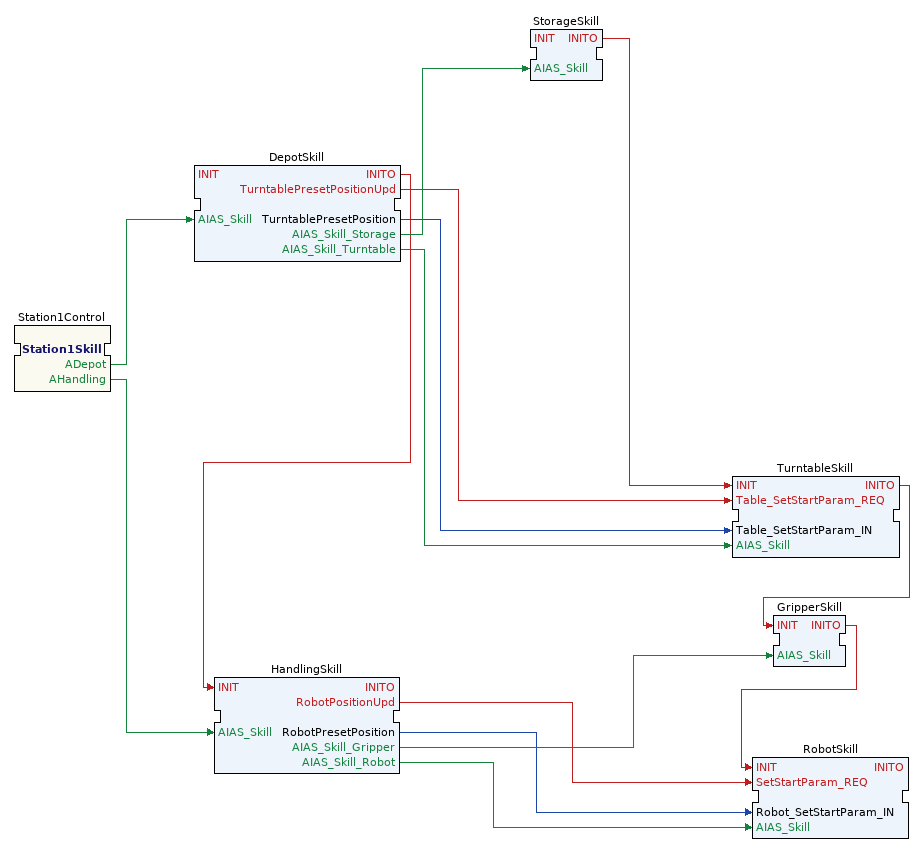
    [picture p24: application VDMA_Station1_SkillbasedControl]
    FBS
      Station1Control : Station1Skill;
    END_FBS
    SUBAPPLICATION StorageSkill
      EVENT_INPUT
        INIT;
      END_EVENT
      EVENT_OUTPUT
        INITO;
      END_EVENT
      SOCKETS
        AIAS_Skill : IAS_Skill;
      END_SOCKETS
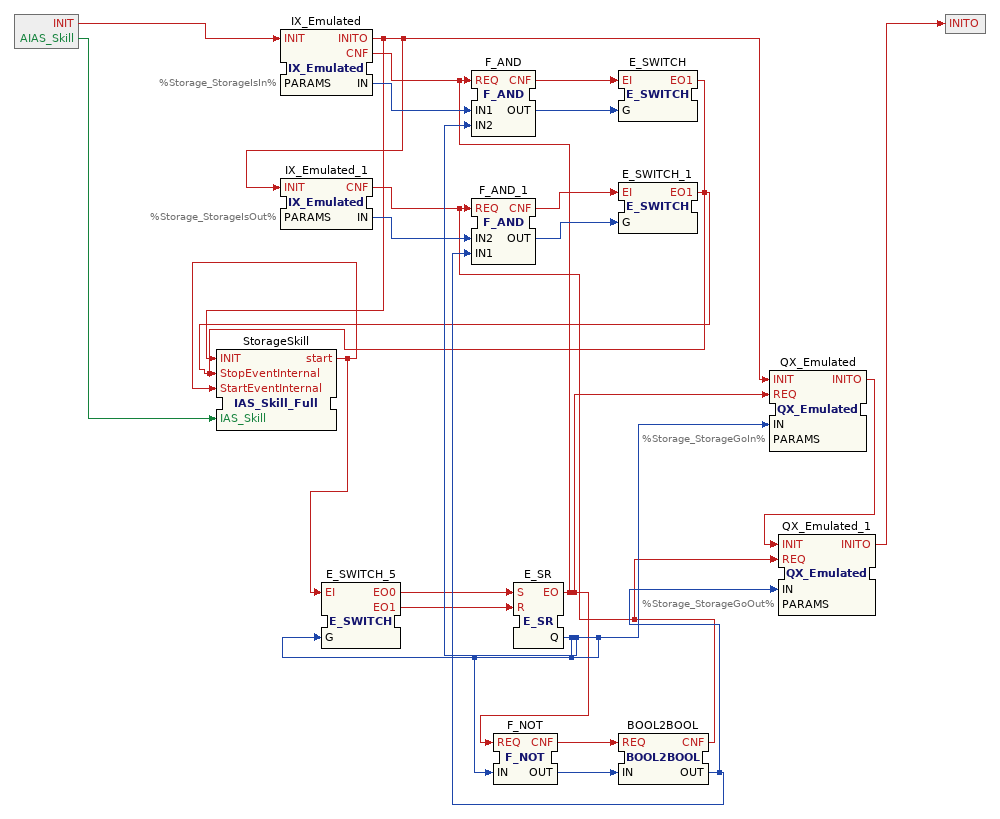
      FBS
        E_SWITCH_5 : E_SWITCH;
        IX_Emulated : IX_Emulated(PARAMS := %Storage_StorageIsIn%);
        F_NOT : F_NOT;
        IX_Emulated_1 : IX_Emulated(PARAMS := %Storage_StorageIsOut%);
        E_SWITCH : E_SWITCH;
        E_SWITCH_1 : E_SWITCH;
        StorageSkill : IAS_Skill_Full;
        F_AND : F_AND;
        BOOL2BOOL : BOOL2BOOL;
        F_AND_1 : F_AND;
        E_SR : E_SR;
        QX_Emulated_1 : QX_Emulated(PARAMS := %Storage_StorageGoOut%);
        QX_Emulated : QX_Emulated(PARAMS := %Storage_StorageGoIn%);
      END_FBS
      EVENT_CONNECTIONS
        StorageSkill.start TO E_SWITCH_5.EI;
        E_SWITCH_5.EO0 TO E_SR.S;
        E_SWITCH_5.EO1 TO E_SR.R;
        IX_Emulated.INITO TO IX_Emulated_1.INIT;
        IX_Emulated.INITO TO StorageSkill.INIT;
        IX_Emulated.CNF TO F_AND.REQ;
        E_SR.EO TO F_NOT.REQ;
        F_NOT.CNF TO BOOL2BOOL.REQ;
        IX_Emulated_1.CNF TO F_AND_1.REQ;
        F_AND.CNF TO E_SWITCH.EI;
        E_SWITCH.EO1 TO StorageSkill.StopEventInternal;
        F_AND_1.CNF TO E_SWITCH_1.EI;
        E_SWITCH_1.EO1 TO StorageSkill.StopEventInternal;
        StorageSkill.start TO StorageSkill.StartEventInternal;
        E_SR.EO TO F_AND.REQ;
        BOOL2BOOL.CNF TO F_AND_1.REQ;
        INIT TO IX_Emulated.INIT;
        QX_Emulated_1.INITO TO INITO;
        IX_Emulated.INITO TO QX_Emulated.INIT;
        QX_Emulated.INITO TO QX_Emulated_1.INIT;
        BOOL2BOOL.CNF TO QX_Emulated_1.REQ;
        E_SR.EO TO QX_Emulated.REQ;
      END_CONNECTIONS
      DATA_CONNECTIONS
        E_SR.Q TO E_SWITCH_5.G;
        IX_Emulated.IN TO F_AND.IN1;
        E_SR.Q TO F_NOT.IN;
        F_NOT.OUT TO BOOL2BOOL.IN;
        IX_Emulated_1.IN TO F_AND_1.IN2;
        F_AND.OUT TO E_SWITCH.G;
        F_AND_1.OUT TO E_SWITCH_1.G;
        E_SR.Q TO F_AND.IN2;
        BOOL2BOOL.OUT TO F_AND_1.IN1;
        E_SR.Q TO QX_Emulated.IN;
        BOOL2BOOL.OUT TO QX_Emulated_1.IN;
      END_CONNECTIONS
      ADAPTER_CONNECTIONS
        AIAS_Skill TO StorageSkill.IAS_Skill;
      END_CONNECTIONS
    END_SUBAPPLICATION
    SUBAPPLICATION TurntableSkill
      EVENT_INPUT
        INIT;
        Table_SetStartParam_REQ;
      END_EVENT
      EVENT_OUTPUT
        INITO;
      END_EVENT
      VAR_INPUT
        Table_SetStartParam_IN : WORD;
      END_VAR
      SOCKETS
        AIAS_Skill : IAS_Skill;
      END_SOCKETS
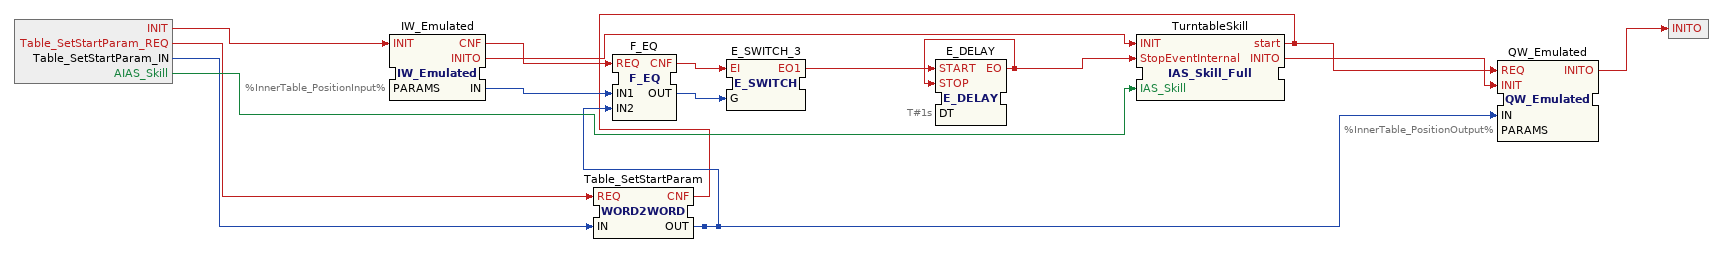
      FBS
        F_EQ : F_EQ;
        E_SWITCH_3 : E_SWITCH;
        Table_SetStartParam : WORD2WORD;
        QW_Emulated : QW_Emulated(PARAMS := %InnerTable_PositionOutput%);
        TurntableSkill : IAS_Skill_Full;
        IW_Emulated : IW_Emulated(PARAMS := %InnerTable_PositionInput%);
        E_DELAY : E_DELAY(DT := T#1s);
      END_FBS
      EVENT_CONNECTIONS
        IW_Emulated.CNF TO F_EQ.REQ;
        TurntableSkill.start TO F_EQ.REQ;
        Table_SetStartParam.CNF TO F_EQ.REQ;
        F_EQ.CNF TO E_SWITCH_3.EI;
        TurntableSkill.start TO QW_Emulated.REQ;
        Table_SetStartParam_REQ TO Table_SetStartParam.REQ;
        INIT TO IW_Emulated.INIT;
        IW_Emulated.INITO TO TurntableSkill.INIT;
        TurntableSkill.INITO TO QW_Emulated.INIT;
        QW_Emulated.INITO TO INITO;
        E_SWITCH_3.EO1 TO E_DELAY.START;
        E_DELAY.EO TO TurntableSkill.StopEventInternal;
        E_DELAY.EO TO E_DELAY.STOP;
      END_CONNECTIONS
      DATA_CONNECTIONS
        IW_Emulated.IN TO F_EQ.IN1;
        Table_SetStartParam.OUT TO F_EQ.IN2;
        F_EQ.OUT TO E_SWITCH_3.G;
        Table_SetStartParam.OUT TO QW_Emulated.IN;
        Table_SetStartParam_IN TO Table_SetStartParam.IN;
      END_CONNECTIONS
      ADAPTER_CONNECTIONS
        AIAS_Skill TO TurntableSkill.IAS_Skill;
      END_CONNECTIONS
    END_SUBAPPLICATION
    SUBAPPLICATION DepotSkill
      EVENT_INPUT
        INIT;
      END_EVENT
      EVENT_OUTPUT
        INITO;
        TurntablePresetPositionUpd;
      END_EVENT
      VAR_OUTPUT
        TurntablePresetPosition : WORD;
      END_VAR
      SOCKETS
        AIAS_Skill : IAS_Skill;
      END_SOCKETS
      PLUGS
        AIAS_Skill_Storage : IAS_Skill;
        AIAS_Skill_Turntable : IAS_Skill;
      END_PLUGS
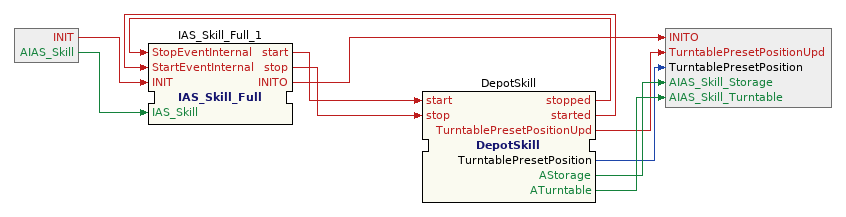
      FBS
        IAS_Skill_Full_1 : IAS_Skill_Full;
        DepotSkill : DepotSkill;
      END_FBS
      EVENT_CONNECTIONS
        DepotSkill.stopped TO IAS_Skill_Full_1.StopEventInternal;
        DepotSkill.started TO IAS_Skill_Full_1.StartEventInternal;
        IAS_Skill_Full_1.start TO DepotSkill.start;
        IAS_Skill_Full_1.stop TO DepotSkill.stop;
        DepotSkill.TurntablePresetPositionUpd TO TurntablePresetPositionUpd;
        INIT TO IAS_Skill_Full_1.INIT;
        IAS_Skill_Full_1.INITO TO INITO;
      END_CONNECTIONS
      DATA_CONNECTIONS
        DepotSkill.TurntablePresetPosition TO TurntablePresetPosition;
      END_CONNECTIONS
      ADAPTER_CONNECTIONS
        AIAS_Skill TO IAS_Skill_Full_1.IAS_Skill;
        DepotSkill.AStorage TO AIAS_Skill_Storage;
        DepotSkill.ATurntable TO AIAS_Skill_Turntable;
      END_CONNECTIONS
    END_SUBAPPLICATION
    SUBAPPLICATION GripperSkill
      EVENT_INPUT
        INIT;
      END_EVENT
      EVENT_OUTPUT
        INITO;
      END_EVENT
      SOCKETS
        AIAS_Skill : IAS_Skill;
      END_SOCKETS
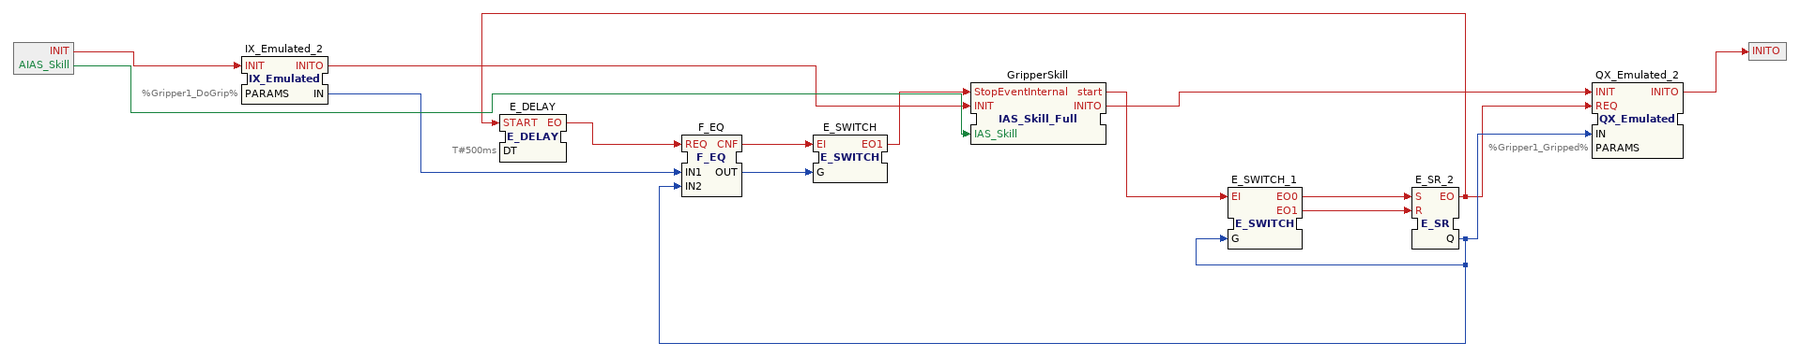
      FBS
        GripperSkill : IAS_Skill_Full;
        F_EQ : F_EQ;
        E_SWITCH_1 : E_SWITCH;
        IX_Emulated_2 : IX_Emulated(PARAMS := %Gripper1_DoGrip%);
        E_DELAY : E_DELAY(DT := T#500ms);
        E_SWITCH : E_SWITCH;
        E_SR_2 : E_SR;
        QX_Emulated_2 : QX_Emulated(PARAMS := %Gripper1_Gripped%);
      END_FBS
      EVENT_CONNECTIONS
        E_SWITCH.EO1 TO GripperSkill.StopEventInternal;
        GripperSkill.start TO E_SWITCH_1.EI;
        E_DELAY.EO TO F_EQ.REQ;
        F_EQ.CNF TO E_SWITCH.EI;
        E_SWITCH_1.EO0 TO E_SR_2.S;
        E_SWITCH_1.EO1 TO E_SR_2.R;
        E_SR_2.EO TO E_DELAY.START;
        INIT TO IX_Emulated_2.INIT;
        IX_Emulated_2.INITO TO GripperSkill.INIT;
        GripperSkill.INITO TO QX_Emulated_2.INIT;
        QX_Emulated_2.INITO TO INITO;
        E_SR_2.EO TO QX_Emulated_2.REQ;
      END_CONNECTIONS
      DATA_CONNECTIONS
        IX_Emulated_2.IN TO F_EQ.IN1;
        E_SR_2.Q TO F_EQ.IN2;
        F_EQ.OUT TO E_SWITCH.G;
        E_SR_2.Q TO E_SWITCH_1.G;
        E_SR_2.Q TO QX_Emulated_2.IN;
      END_CONNECTIONS
      ADAPTER_CONNECTIONS
        AIAS_Skill TO GripperSkill.IAS_Skill;
      END_CONNECTIONS
    END_SUBAPPLICATION
    SUBAPPLICATION HandlingSkill
      EVENT_INPUT
        INIT;
      END_EVENT
      EVENT_OUTPUT
        INITO;
        RobotPositionUpd;
      END_EVENT
      VAR_OUTPUT
        RobotPresetPosition : WORD;
      END_VAR
      SOCKETS
        AIAS_Skill : IAS_Skill;
      END_SOCKETS
      PLUGS
        AIAS_Skill_Gripper : IAS_Skill;
        AIAS_Skill_Robot : IAS_Skill;
      END_PLUGS
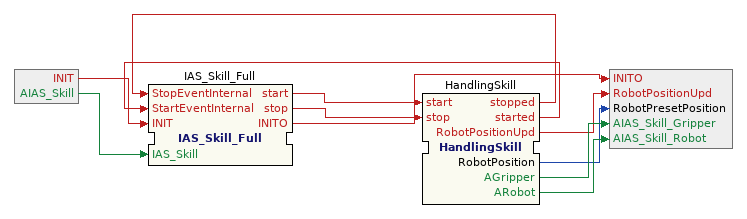
      FBS
        IAS_Skill_Full : IAS_Skill_Full;
        HandlingSkill : HandlingSkill;
      END_FBS
      EVENT_CONNECTIONS
        HandlingSkill.stopped TO IAS_Skill_Full.StopEventInternal;
        HandlingSkill.started TO IAS_Skill_Full.StartEventInternal;
        IAS_Skill_Full.start TO HandlingSkill.start;
        IAS_Skill_Full.stop TO HandlingSkill.stop;
        HandlingSkill.RobotPositionUpd TO RobotPositionUpd;
        INIT TO IAS_Skill_Full.INIT;
        IAS_Skill_Full.INITO TO INITO;
      END_CONNECTIONS
      DATA_CONNECTIONS
        HandlingSkill.RobotPosition TO RobotPresetPosition;
      END_CONNECTIONS
      ADAPTER_CONNECTIONS
        AIAS_Skill TO IAS_Skill_Full.IAS_Skill;
        HandlingSkill.AGripper TO AIAS_Skill_Gripper;
        HandlingSkill.ARobot TO AIAS_Skill_Robot;
      END_CONNECTIONS
    END_SUBAPPLICATION
    SUBAPPLICATION RobotSkill
      EVENT_INPUT
        INIT;
        SetStartParam_REQ;
      END_EVENT
      EVENT_OUTPUT
        INITO;
      END_EVENT
      VAR_INPUT
        Robot_SetStartParam_IN : WORD;
      END_VAR
      SOCKETS
        AIAS_Skill : IAS_Skill;
      END_SOCKETS
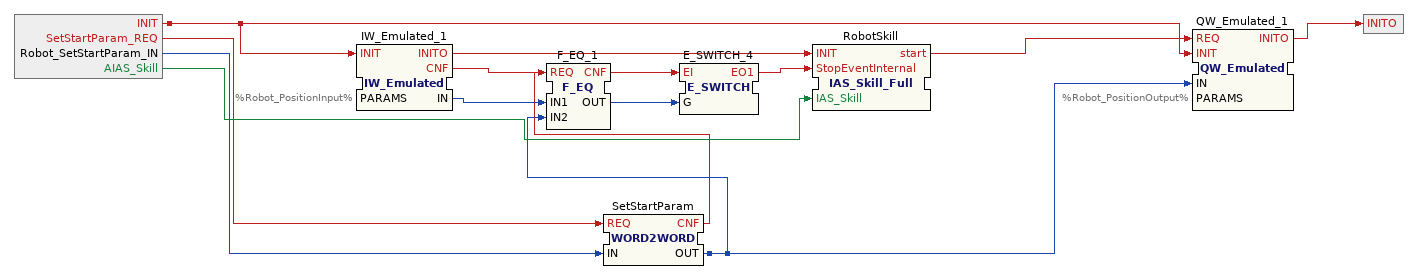
      FBS
        RobotSkill : IAS_Skill_Full;
        IW_Emulated_1 : IW_Emulated(PARAMS := %Robot_PositionInput%);
        E_SWITCH_4 : E_SWITCH;
        F_EQ_1 : F_EQ;
        QW_Emulated_1 : QW_Emulated(PARAMS := %Robot_PositionOutput%);
        SetStartParam : WORD2WORD;
      END_FBS
      EVENT_CONNECTIONS
        IW_Emulated_1.INITO TO RobotSkill.INIT;
        E_SWITCH_4.EO1 TO RobotSkill.StopEventInternal;
        RobotSkill.start TO QW_Emulated_1.REQ;
        IW_Emulated_1.CNF TO F_EQ_1.REQ;
        F_EQ_1.CNF TO E_SWITCH_4.EI;
        SetStartParam.CNF TO F_EQ_1.REQ;
        INIT TO QW_Emulated_1.INIT;
        QW_Emulated_1.INITO TO INITO;
        SetStartParam_REQ TO SetStartParam.REQ;
        INIT TO IW_Emulated_1.INIT;
      END_CONNECTIONS
      DATA_CONNECTIONS
        IW_Emulated_1.IN TO F_EQ_1.IN1;
        F_EQ_1.OUT TO E_SWITCH_4.G;
        SetStartParam.OUT TO F_EQ_1.IN2;
        SetStartParam.OUT TO QW_Emulated_1.IN;
        Robot_SetStartParam_IN TO SetStartParam.IN;
      END_CONNECTIONS
      ADAPTER_CONNECTIONS
        AIAS_Skill TO RobotSkill.IAS_Skill;
      END_CONNECTIONS
    END_SUBAPPLICATION
    EVENT_CONNECTIONS
      DepotSkill.TurntablePresetPositionUpd TO TurntableSkill.Table_SetStartParam_REQ;
      StorageSkill.INITO TO TurntableSkill.INIT;
      TurntableSkill.INITO TO GripperSkill.INIT;
      DepotSkill.INITO TO HandlingSkill.INIT;
      HandlingSkill.RobotPositionUpd TO RobotSkill.SetStartParam_REQ;
      GripperSkill.INITO TO RobotSkill.INIT;
    END_CONNECTIONS
    DATA_CONNECTIONS
      DepotSkill.TurntablePresetPosition TO TurntableSkill.Table_SetStartParam_IN;
      HandlingSkill.RobotPresetPosition TO RobotSkill.Robot_SetStartParam_IN;
    END_CONNECTIONS
    ADAPTER_CONNECTIONS
      Station1Control.ADepot TO DepotSkill.AIAS_Skill;
      DepotSkill.AIAS_Skill_Storage TO StorageSkill.AIAS_Skill;
      DepotSkill.AIAS_Skill_Turntable TO TurntableSkill.AIAS_Skill;
      Station1Control.AHandling TO HandlingSkill.AIAS_Skill;
      HandlingSkill.AIAS_Skill_Gripper TO GripperSkill.AIAS_Skill;
      HandlingSkill.AIAS_Skill_Robot TO RobotSkill.AIAS_Skill;
    END_CONNECTIONS
  END_APPLICATION
  APPLICATION VDMA_Station1_CodeGenTemplate
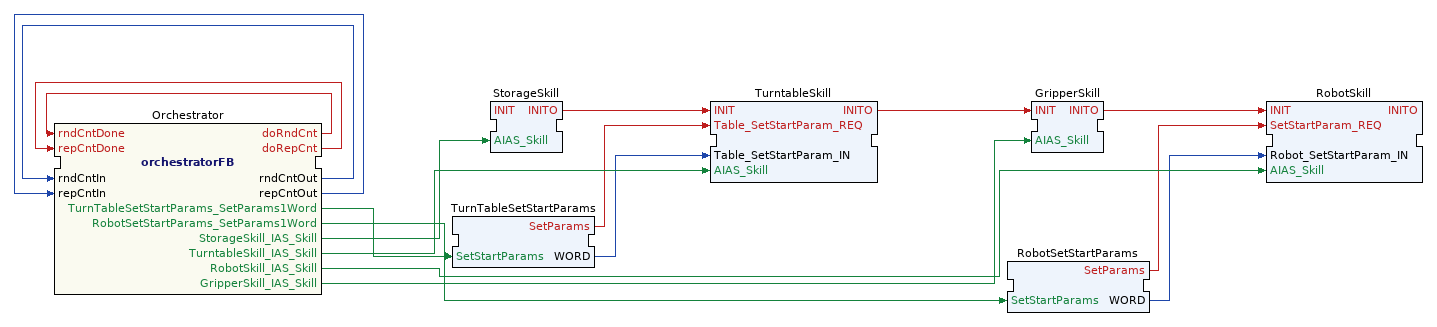
    FBS
      Orchestrator : orchestratorFB;
    END_FBS
    SUBAPPLICATION TurnTableSetStartParams
      EVENT_OUTPUT
        SetParams;
      END_EVENT
      VAR_OUTPUT
        WORD : WORD;
      END_VAR
      SOCKETS
        SetStartParams : SetParams1Word;
      END_SOCKETS
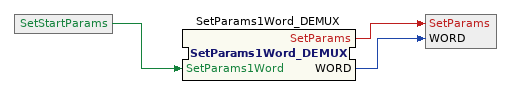
      FBS
        SetParams1Word_DEMUX : SetParams1Word_DEMUX;
      END_FBS
      EVENT_CONNECTIONS
        SetParams1Word_DEMUX.SetParams TO SetParams;
      END_CONNECTIONS
      DATA_CONNECTIONS
        SetParams1Word_DEMUX.WORD TO WORD;
      END_CONNECTIONS
      ADAPTER_CONNECTIONS
        SetStartParams TO SetParams1Word_DEMUX.SetParams1Word;
      END_CONNECTIONS
    END_SUBAPPLICATION
    SUBAPPLICATION RobotSetStartParams
      EVENT_OUTPUT
        SetParams;
      END_EVENT
      VAR_OUTPUT
        WORD : WORD;
      END_VAR
      SOCKETS
        SetStartParams : SetParams1Word;
      END_SOCKETS
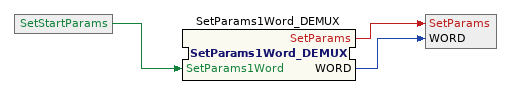
      FBS
        SetParams1Word_DEMUX : SetParams1Word_DEMUX;
      END_FBS
      EVENT_CONNECTIONS
        SetParams1Word_DEMUX.SetParams TO SetParams;
      END_CONNECTIONS
      DATA_CONNECTIONS
        SetParams1Word_DEMUX.WORD TO WORD;
      END_CONNECTIONS
      ADAPTER_CONNECTIONS
        SetStartParams TO SetParams1Word_DEMUX.SetParams1Word;
      END_CONNECTIONS
    END_SUBAPPLICATION
    SUBAPPLICATION TurntableSkill
      EVENT_INPUT
        INIT;
        Table_SetStartParam_REQ;
      END_EVENT
      EVENT_OUTPUT
        INITO;
      END_EVENT
      VAR_INPUT
        Table_SetStartParam_IN : WORD;
      END_VAR
      SOCKETS
        AIAS_Skill : IAS_Skill;
      END_SOCKETS
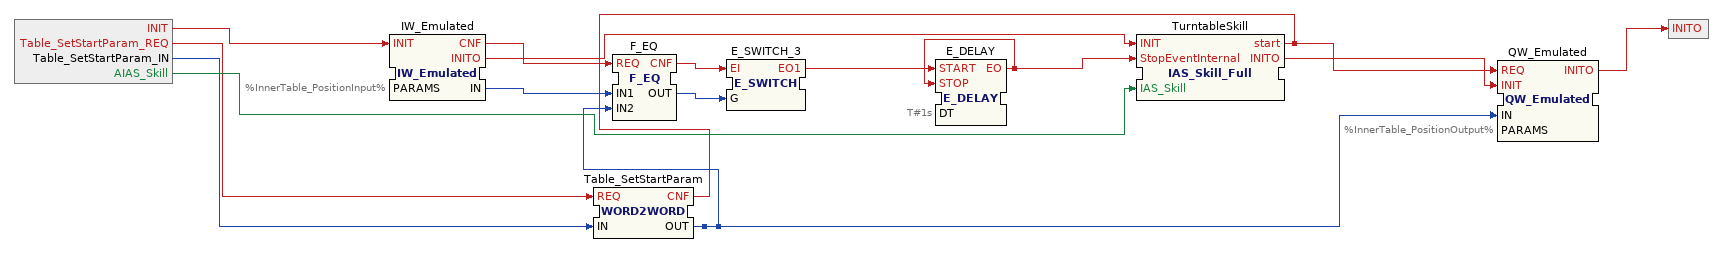
      FBS
        F_EQ : F_EQ;
        E_SWITCH_3 : E_SWITCH;
        Table_SetStartParam : WORD2WORD;
        QW_Emulated : QW_Emulated(PARAMS := %InnerTable_PositionOutput%);
        TurntableSkill : IAS_Skill_Full;
        IW_Emulated : IW_Emulated(PARAMS := %InnerTable_PositionInput%);
        E_DELAY : E_DELAY(DT := T#1s);
      END_FBS
      EVENT_CONNECTIONS
        IW_Emulated.CNF TO F_EQ.REQ;
        TurntableSkill.start TO F_EQ.REQ;
        Table_SetStartParam.CNF TO F_EQ.REQ;
        F_EQ.CNF TO E_SWITCH_3.EI;
        TurntableSkill.start TO QW_Emulated.REQ;
        Table_SetStartParam_REQ TO Table_SetStartParam.REQ;
        INIT TO IW_Emulated.INIT;
        IW_Emulated.INITO TO TurntableSkill.INIT;
        TurntableSkill.INITO TO QW_Emulated.INIT;
        QW_Emulated.INITO TO INITO;
        E_SWITCH_3.EO1 TO E_DELAY.START;
        E_DELAY.EO TO TurntableSkill.StopEventInternal;
        E_DELAY.EO TO E_DELAY.STOP;
      END_CONNECTIONS
      DATA_CONNECTIONS
        IW_Emulated.IN TO F_EQ.IN1;
        Table_SetStartParam.OUT TO F_EQ.IN2;
        F_EQ.OUT TO E_SWITCH_3.G;
        Table_SetStartParam.OUT TO QW_Emulated.IN;
        Table_SetStartParam_IN TO Table_SetStartParam.IN;
      END_CONNECTIONS
      ADAPTER_CONNECTIONS
        AIAS_Skill TO TurntableSkill.IAS_Skill;
      END_CONNECTIONS
    END_SUBAPPLICATION
    SUBAPPLICATION GripperSkill
      EVENT_INPUT
        INIT;
      END_EVENT
      EVENT_OUTPUT
        INITO;
      END_EVENT
      SOCKETS
        AIAS_Skill : IAS_Skill;
      END_SOCKETS
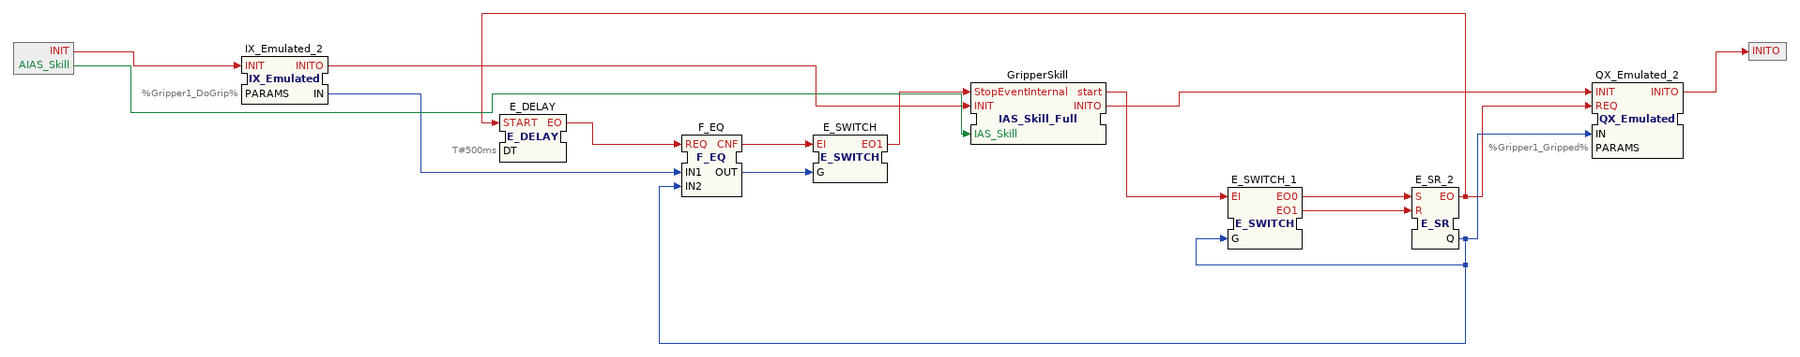
      FBS
        GripperSkill : IAS_Skill_Full;
        F_EQ : F_EQ;
        E_SWITCH_1 : E_SWITCH;
        IX_Emulated_2 : IX_Emulated(PARAMS := %Gripper1_DoGrip%);
        E_DELAY : E_DELAY(DT := T#500ms);
        E_SWITCH : E_SWITCH;
        E_SR_2 : E_SR;
        QX_Emulated_2 : QX_Emulated(PARAMS := %Gripper1_Gripped%);
      END_FBS
      EVENT_CONNECTIONS
        E_SWITCH.EO1 TO GripperSkill.StopEventInternal;
        GripperSkill.start TO E_SWITCH_1.EI;
        E_DELAY.EO TO F_EQ.REQ;
        F_EQ.CNF TO E_SWITCH.EI;
        E_SWITCH_1.EO0 TO E_SR_2.S;
        E_SWITCH_1.EO1 TO E_SR_2.R;
        E_SR_2.EO TO E_DELAY.START;
        INIT TO IX_Emulated_2.INIT;
        IX_Emulated_2.INITO TO GripperSkill.INIT;
        GripperSkill.INITO TO QX_Emulated_2.INIT;
        QX_Emulated_2.INITO TO INITO;
        E_SR_2.EO TO QX_Emulated_2.REQ;
      END_CONNECTIONS
      DATA_CONNECTIONS
        IX_Emulated_2.IN TO F_EQ.IN1;
        E_SR_2.Q TO F_EQ.IN2;
        F_EQ.OUT TO E_SWITCH.G;
        E_SR_2.Q TO E_SWITCH_1.G;
        E_SR_2.Q TO QX_Emulated_2.IN;
      END_CONNECTIONS
      ADAPTER_CONNECTIONS
        AIAS_Skill TO GripperSkill.IAS_Skill;
      END_CONNECTIONS
    END_SUBAPPLICATION
    SUBAPPLICATION RobotSkill
      EVENT_INPUT
        INIT;
        SetStartParam_REQ;
      END_EVENT
      EVENT_OUTPUT
        INITO;
      END_EVENT
      VAR_INPUT
        Robot_SetStartParam_IN : WORD;
      END_VAR
      SOCKETS
        AIAS_Skill : IAS_Skill;
      END_SOCKETS
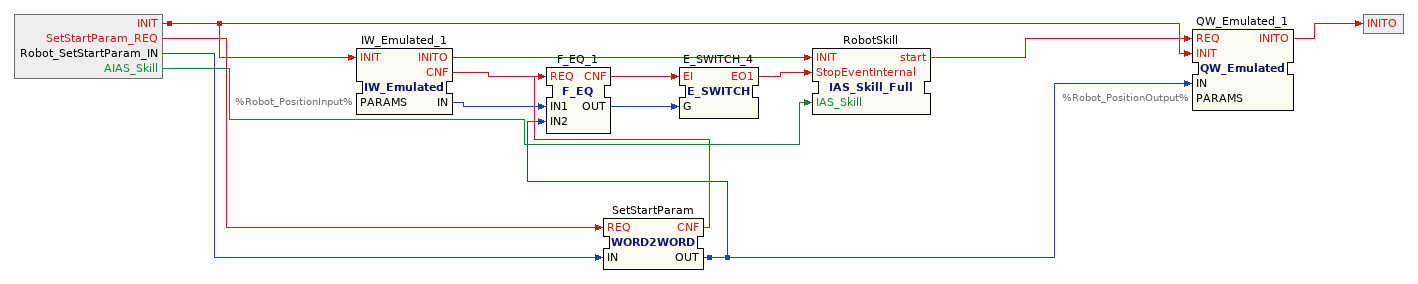
      FBS
        RobotSkill : IAS_Skill_Full;
        IW_Emulated_1 : IW_Emulated(PARAMS := %Robot_PositionInput%);
        E_SWITCH_4 : E_SWITCH;
        F_EQ_1 : F_EQ;
        QW_Emulated_1 : QW_Emulated(PARAMS := %Robot_PositionOutput%);
        SetStartParam : WORD2WORD;
      END_FBS
      EVENT_CONNECTIONS
        IW_Emulated_1.INITO TO RobotSkill.INIT;
        E_SWITCH_4.EO1 TO RobotSkill.StopEventInternal;
        RobotSkill.start TO QW_Emulated_1.REQ;
        IW_Emulated_1.CNF TO F_EQ_1.REQ;
        F_EQ_1.CNF TO E_SWITCH_4.EI;
        SetStartParam.CNF TO F_EQ_1.REQ;
        INIT TO IW_Emulated_1.INIT;
        SetStartParam_REQ TO SetStartParam.REQ;
        QW_Emulated_1.INITO TO INITO;
        INIT TO QW_Emulated_1.INIT;
      END_CONNECTIONS
      DATA_CONNECTIONS
        IW_Emulated_1.IN TO F_EQ_1.IN1;
        F_EQ_1.OUT TO E_SWITCH_4.G;
        SetStartParam.OUT TO F_EQ_1.IN2;
        SetStartParam.OUT TO QW_Emulated_1.IN;
        Robot_SetStartParam_IN TO SetStartParam.IN;
      END_CONNECTIONS
      ADAPTER_CONNECTIONS
        AIAS_Skill TO RobotSkill.IAS_Skill;
      END_CONNECTIONS
    END_SUBAPPLICATION
    SUBAPPLICATION StorageSkill
      EVENT_INPUT
        INIT;
      END_EVENT
      EVENT_OUTPUT
        INITO;
      END_EVENT
      SOCKETS
        AIAS_Skill : IAS_Skill;
      END_SOCKETS
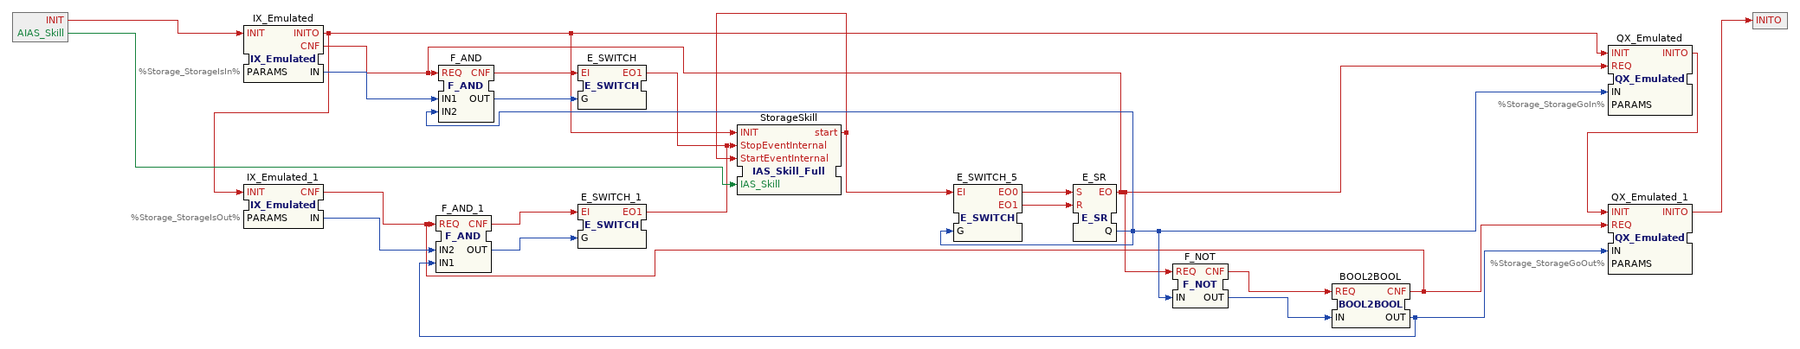
      FBS
        E_SWITCH_5 : E_SWITCH;
        IX_Emulated : IX_Emulated(PARAMS := %Storage_StorageIsIn%);
        F_NOT : F_NOT;
        IX_Emulated_1 : IX_Emulated(PARAMS := %Storage_StorageIsOut%);
        E_SWITCH : E_SWITCH;
        E_SWITCH_1 : E_SWITCH;
        StorageSkill : IAS_Skill_Full;
        F_AND : F_AND;
        BOOL2BOOL : BOOL2BOOL;
        F_AND_1 : F_AND;
        E_SR : E_SR;
        QX_Emulated_1 : QX_Emulated(PARAMS := %Storage_StorageGoOut%);
        QX_Emulated : QX_Emulated(PARAMS := %Storage_StorageGoIn%);
      END_FBS
      EVENT_CONNECTIONS
        StorageSkill.start TO E_SWITCH_5.EI;
        E_SWITCH_5.EO0 TO E_SR.S;
        E_SWITCH_5.EO1 TO E_SR.R;
        IX_Emulated.INITO TO IX_Emulated_1.INIT;
        IX_Emulated.INITO TO StorageSkill.INIT;
        IX_Emulated.CNF TO F_AND.REQ;
        E_SR.EO TO F_NOT.REQ;
        F_NOT.CNF TO BOOL2BOOL.REQ;
        IX_Emulated_1.CNF TO F_AND_1.REQ;
        F_AND.CNF TO E_SWITCH.EI;
        E_SWITCH.EO1 TO StorageSkill.StopEventInternal;
        F_AND_1.CNF TO E_SWITCH_1.EI;
        E_SWITCH_1.EO1 TO StorageSkill.StopEventInternal;
        StorageSkill.start TO StorageSkill.StartEventInternal;
        E_SR.EO TO F_AND.REQ;
        BOOL2BOOL.CNF TO F_AND_1.REQ;
        INIT TO IX_Emulated.INIT;
        QX_Emulated_1.INITO TO INITO;
        IX_Emulated.INITO TO QX_Emulated.INIT;
        QX_Emulated.INITO TO QX_Emulated_1.INIT;
        BOOL2BOOL.CNF TO QX_Emulated_1.REQ;
        E_SR.EO TO QX_Emulated.REQ;
      END_CONNECTIONS
      DATA_CONNECTIONS
        E_SR.Q TO E_SWITCH_5.G;
        IX_Emulated.IN TO F_AND.IN1;
        E_SR.Q TO F_NOT.IN;
        F_NOT.OUT TO BOOL2BOOL.IN;
        IX_Emulated_1.IN TO F_AND_1.IN2;
        F_AND.OUT TO E_SWITCH.G;
        F_AND_1.OUT TO E_SWITCH_1.G;
        E_SR.Q TO F_AND.IN2;
        BOOL2BOOL.OUT TO F_AND_1.IN1;
        E_SR.Q TO QX_Emulated.IN;
        BOOL2BOOL.OUT TO QX_Emulated_1.IN;
      END_CONNECTIONS
      ADAPTER_CONNECTIONS
        AIAS_Skill TO StorageSkill.IAS_Skill;
      END_CONNECTIONS
    END_SUBAPPLICATION
    EVENT_CONNECTIONS
      Orchestrator.doRndCnt TO Orchestrator.rndCntDone; (* Self loop *)
      Orchestrator.doRepCnt TO Orchestrator.repCntDone; (* Self loop *)
      StorageSkill.INITO TO TurntableSkill.INIT;
      GripperSkill.INITO TO RobotSkill.INIT;
      TurntableSkill.INITO TO GripperSkill.INIT;
      TurnTableSetStartParams.SetParams TO TurntableSkill.Table_SetStartParam_REQ;
      RobotSetStartParams.SetParams TO RobotSkill.SetStartParam_REQ;
    END_CONNECTIONS
    DATA_CONNECTIONS
      Orchestrator.rndCntOut TO Orchestrator.rndCntIn; (* Self loop *)
      Orchestrator.repCntOut TO Orchestrator.repCntIn; (* Self loop *)
      TurnTableSetStartParams.WORD TO TurntableSkill.Table_SetStartParam_IN;
      RobotSetStartParams.WORD TO RobotSkill.Robot_SetStartParam_IN;
    END_CONNECTIONS
    ADAPTER_CONNECTIONS
      Orchestrator.TurnTableSetStartParams_SetParams1Word TO TurnTableSetStartParams.SetStartParams;
      Orchestrator.RobotSetStartParams_SetParams1Word TO RobotSetStartParams.SetStartParams;
      Orchestrator.StorageSkill_IAS_Skill TO StorageSkill.AIAS_Skill;
      Orchestrator.TurntableSkill_IAS_Skill TO TurntableSkill.AIAS_Skill;
      Orchestrator.RobotSkill_IAS_Skill TO RobotSkill.AIAS_Skill;
      Orchestrator.GripperSkill_IAS_Skill TO GripperSkill.AIAS_Skill;
    END_CONNECTIONS
  END_APPLICATION
  APPLICATION VDMA_Station1_CodeGenControl
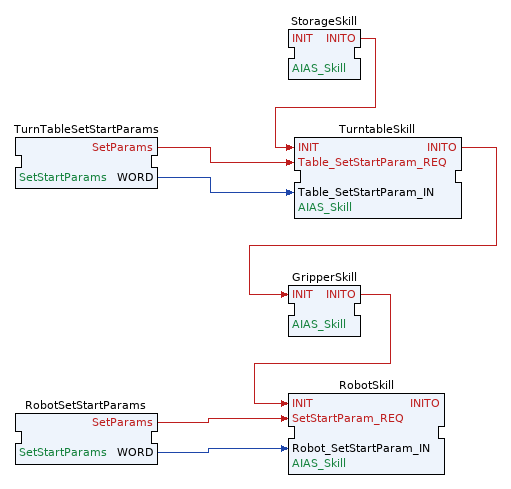
    SUBAPPLICATION StorageSkill
      EVENT_INPUT
        INIT;
      END_EVENT
      EVENT_OUTPUT
        INITO;
      END_EVENT
      SOCKETS
        AIAS_Skill : IAS_Skill;
      END_SOCKETS
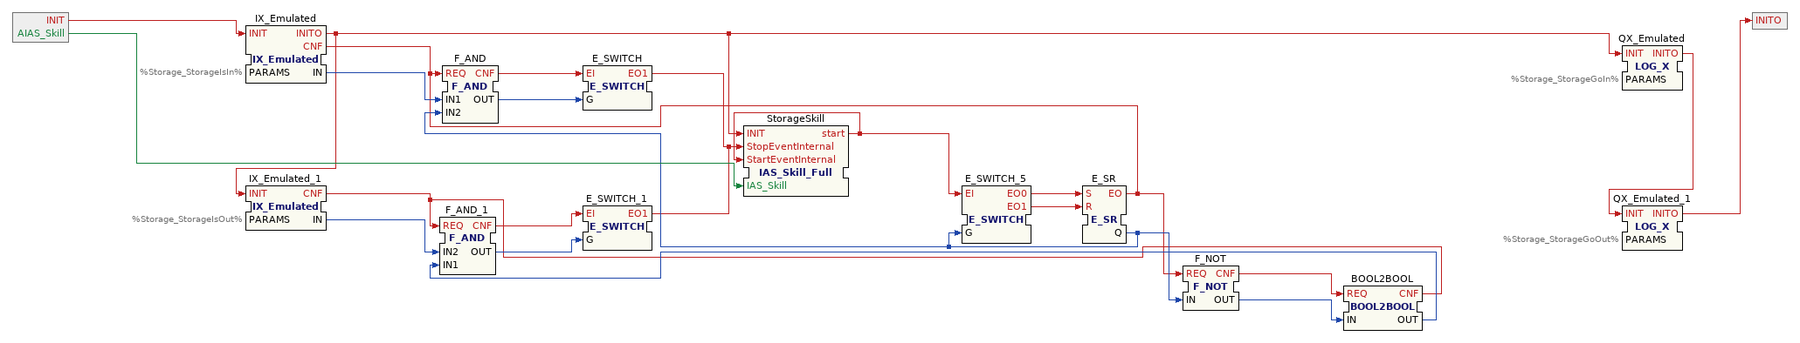
      FBS
        E_SWITCH_5 : E_SWITCH;
        IX_Emulated : IX_Emulated(PARAMS := %Storage_StorageIsIn%);
        QX_Emulated_1 : LOG_X(PARAMS := %Storage_StorageGoOut%);
        F_NOT : F_NOT;
        QX_Emulated : LOG_X(PARAMS := %Storage_StorageGoIn%);
        IX_Emulated_1 : IX_Emulated(PARAMS := %Storage_StorageIsOut%);
        E_SWITCH : E_SWITCH;
        E_SWITCH_1 : E_SWITCH;
        StorageSkill : IAS_Skill_Full;
        F_AND : F_AND;
        BOOL2BOOL : BOOL2BOOL;
        F_AND_1 : F_AND;
        E_SR : E_SR;
      END_FBS
      EVENT_CONNECTIONS
        StorageSkill.start TO E_SWITCH_5.EI;
        E_SWITCH_5.EO0 TO E_SR.S;
        E_SWITCH_5.EO1 TO E_SR.R;
        IX_Emulated.INITO TO IX_Emulated_1.INIT;
        IX_Emulated.INITO TO QX_Emulated.INIT;
        IX_Emulated.INITO TO StorageSkill.INIT;
        IX_Emulated.CNF TO F_AND.REQ;
        QX_Emulated.INITO TO QX_Emulated_1.INIT;
        E_SR.EO TO F_NOT.REQ;
        F_NOT.CNF TO BOOL2BOOL.REQ;
        IX_Emulated_1.CNF TO F_AND_1.REQ;
        F_AND.CNF TO E_SWITCH.EI;
        E_SWITCH.EO1 TO StorageSkill.StopEventInternal;
        F_AND_1.CNF TO E_SWITCH_1.EI;
        E_SWITCH_1.EO1 TO StorageSkill.StopEventInternal;
        StorageSkill.start TO StorageSkill.StartEventInternal;
        E_SR.EO TO F_AND.REQ;
        BOOL2BOOL.CNF TO F_AND_1.REQ;
        INIT TO IX_Emulated.INIT;
        QX_Emulated_1.INITO TO INITO;
      END_CONNECTIONS
      DATA_CONNECTIONS
        E_SR.Q TO E_SWITCH_5.G;
        IX_Emulated.IN TO F_AND.IN1;
        E_SR.Q TO F_NOT.IN;
        F_NOT.OUT TO BOOL2BOOL.IN;
        IX_Emulated_1.IN TO F_AND_1.IN2;
        F_AND.OUT TO E_SWITCH.G;
        F_AND_1.OUT TO E_SWITCH_1.G;
        E_SR.Q TO F_AND.IN2;
        BOOL2BOOL.OUT TO F_AND_1.IN1;
      END_CONNECTIONS
      ADAPTER_CONNECTIONS
        AIAS_Skill TO StorageSkill.IAS_Skill;
      END_CONNECTIONS
    END_SUBAPPLICATION
    SUBAPPLICATION TurntableSkill
      EVENT_INPUT
        INIT;
        Table_SetStartParam_REQ;
      END_EVENT
      EVENT_OUTPUT
        INITO;
      END_EVENT
      VAR_INPUT
        Table_SetStartParam_IN : WORD;
      END_VAR
      SOCKETS
        AIAS_Skill : IAS_Skill;
      END_SOCKETS
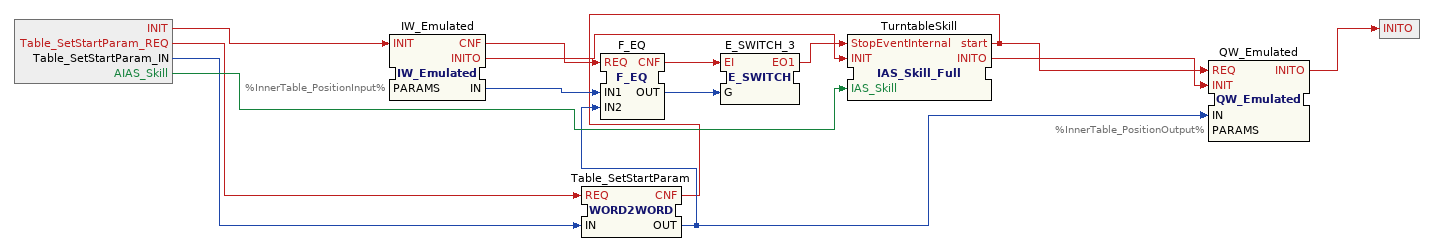
      FBS
        F_EQ : F_EQ;
        E_SWITCH_3 : E_SWITCH;
        Table_SetStartParam : WORD2WORD;
        QW_Emulated : QW_Emulated(PARAMS := %InnerTable_PositionOutput%);
        TurntableSkill : IAS_Skill_Full;
        IW_Emulated : IW_Emulated(PARAMS := %InnerTable_PositionInput%);
      END_FBS
      EVENT_CONNECTIONS
        IW_Emulated.CNF TO F_EQ.REQ;
        TurntableSkill.start TO F_EQ.REQ;
        Table_SetStartParam.CNF TO F_EQ.REQ;
        F_EQ.CNF TO E_SWITCH_3.EI;
        E_SWITCH_3.EO1 TO TurntableSkill.StopEventInternal;
        TurntableSkill.start TO QW_Emulated.REQ;
        INIT TO IW_Emulated.INIT;
        IW_Emulated.INITO TO TurntableSkill.INIT;
        TurntableSkill.INITO TO QW_Emulated.INIT;
        QW_Emulated.INITO TO INITO;
        Table_SetStartParam_REQ TO Table_SetStartParam.REQ;
      END_CONNECTIONS
      DATA_CONNECTIONS
        IW_Emulated.IN TO F_EQ.IN1;
        Table_SetStartParam.OUT TO F_EQ.IN2;
        F_EQ.OUT TO E_SWITCH_3.G;
        Table_SetStartParam.OUT TO QW_Emulated.IN;
        Table_SetStartParam_IN TO Table_SetStartParam.IN;
      END_CONNECTIONS
      ADAPTER_CONNECTIONS
        AIAS_Skill TO TurntableSkill.IAS_Skill;
      END_CONNECTIONS
    END_SUBAPPLICATION
    SUBAPPLICATION GripperSkill
      EVENT_INPUT
        INIT;
      END_EVENT
      EVENT_OUTPUT
        INITO;
      END_EVENT
      SOCKETS
        AIAS_Skill : IAS_Skill;
      END_SOCKETS
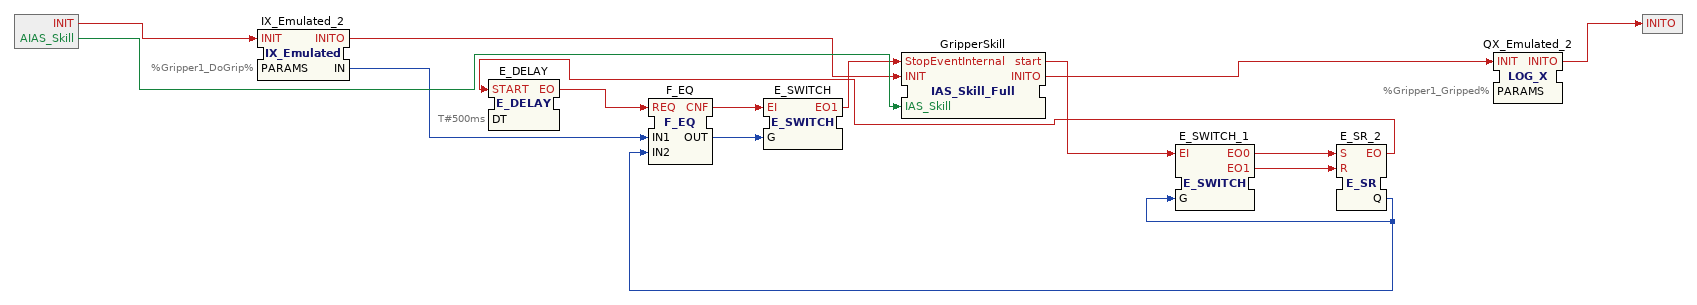
      FBS
        GripperSkill : IAS_Skill_Full;
        F_EQ : F_EQ;
        E_SWITCH_1 : E_SWITCH;
        IX_Emulated_2 : IX_Emulated(PARAMS := %Gripper1_DoGrip%);
        QX_Emulated_2 : LOG_X(PARAMS := %Gripper1_Gripped%);
        E_DELAY : E_DELAY(DT := T#500ms);
        E_SWITCH : E_SWITCH;
        E_SR_2 : E_SR;
      END_FBS
      EVENT_CONNECTIONS
        E_SWITCH.EO1 TO GripperSkill.StopEventInternal;
        GripperSkill.start TO E_SWITCH_1.EI;
        E_DELAY.EO TO F_EQ.REQ;
        F_EQ.CNF TO E_SWITCH.EI;
        E_SWITCH_1.EO0 TO E_SR_2.S;
        E_SWITCH_1.EO1 TO E_SR_2.R;
        E_SR_2.EO TO E_DELAY.START;
        INIT TO IX_Emulated_2.INIT;
        IX_Emulated_2.INITO TO GripperSkill.INIT;
        GripperSkill.INITO TO QX_Emulated_2.INIT;
        QX_Emulated_2.INITO TO INITO;
      END_CONNECTIONS
      DATA_CONNECTIONS
        IX_Emulated_2.IN TO F_EQ.IN1;
        E_SR_2.Q TO F_EQ.IN2;
        F_EQ.OUT TO E_SWITCH.G;
        E_SR_2.Q TO E_SWITCH_1.G;
      END_CONNECTIONS
      ADAPTER_CONNECTIONS
        AIAS_Skill TO GripperSkill.IAS_Skill;
      END_CONNECTIONS
    END_SUBAPPLICATION
    SUBAPPLICATION RobotSkill
      EVENT_INPUT
        INIT;
        SetStartParam_REQ;
      END_EVENT
      EVENT_OUTPUT
        INITO;
      END_EVENT
      VAR_INPUT
        Robot_SetStartParam_IN : WORD;
      END_VAR
      SOCKETS
        AIAS_Skill : IAS_Skill;
      END_SOCKETS
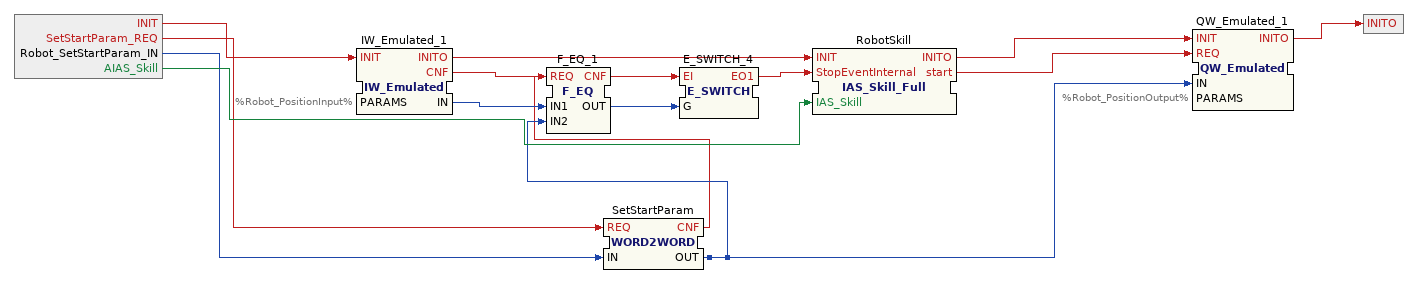
      FBS
        RobotSkill : IAS_Skill_Full;
        IW_Emulated_1 : IW_Emulated(PARAMS := %Robot_PositionInput%);
        E_SWITCH_4 : E_SWITCH;
        F_EQ_1 : F_EQ;
        QW_Emulated_1 : QW_Emulated(PARAMS := %Robot_PositionOutput%);
        SetStartParam : WORD2WORD;
      END_FBS
      EVENT_CONNECTIONS
        IW_Emulated_1.INITO TO RobotSkill.INIT;
        E_SWITCH_4.EO1 TO RobotSkill.StopEventInternal;
        RobotSkill.INITO TO QW_Emulated_1.INIT;
        RobotSkill.start TO QW_Emulated_1.REQ;
        IW_Emulated_1.CNF TO F_EQ_1.REQ;
        F_EQ_1.CNF TO E_SWITCH_4.EI;
        SetStartParam.CNF TO F_EQ_1.REQ;
        INIT TO IW_Emulated_1.INIT;
        SetStartParam_REQ TO SetStartParam.REQ;
        QW_Emulated_1.INITO TO INITO;
      END_CONNECTIONS
      DATA_CONNECTIONS
        IW_Emulated_1.IN TO F_EQ_1.IN1;
        F_EQ_1.OUT TO E_SWITCH_4.G;
        SetStartParam.OUT TO F_EQ_1.IN2;
        SetStartParam.OUT TO QW_Emulated_1.IN;
        Robot_SetStartParam_IN TO SetStartParam.IN;
      END_CONNECTIONS
      ADAPTER_CONNECTIONS
        AIAS_Skill TO RobotSkill.IAS_Skill;
      END_CONNECTIONS
    END_SUBAPPLICATION
    SUBAPPLICATION TurnTableSetStartParams
      EVENT_OUTPUT
        SetParams;
      END_EVENT
      VAR_OUTPUT
        WORD : WORD;
      END_VAR
      SOCKETS
        SetStartParams : SetParams1Word;
      END_SOCKETS
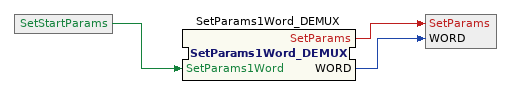
      FBS
        SetParams1Word_DEMUX : SetParams1Word_DEMUX;
      END_FBS
      EVENT_CONNECTIONS
        SetParams1Word_DEMUX.SetParams TO SetParams;
      END_CONNECTIONS
      DATA_CONNECTIONS
        SetParams1Word_DEMUX.WORD TO WORD;
      END_CONNECTIONS
      ADAPTER_CONNECTIONS
        SetStartParams TO SetParams1Word_DEMUX.SetParams1Word;
      END_CONNECTIONS
    END_SUBAPPLICATION
    SUBAPPLICATION RobotSetStartParams
      EVENT_OUTPUT
        SetParams;
      END_EVENT
      VAR_OUTPUT
        WORD : WORD;
      END_VAR
      SOCKETS
        SetStartParams : SetParams1Word;
      END_SOCKETS
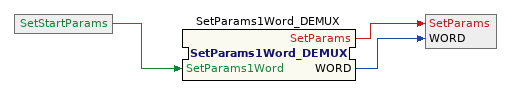
      FBS
        SetParams1Word_DEMUX : SetParams1Word_DEMUX;
      END_FBS
      EVENT_CONNECTIONS
        SetParams1Word_DEMUX.SetParams TO SetParams;
      END_CONNECTIONS
      DATA_CONNECTIONS
        SetParams1Word_DEMUX.WORD TO WORD;
      END_CONNECTIONS
      ADAPTER_CONNECTIONS
        SetStartParams TO SetParams1Word_DEMUX.SetParams1Word;
      END_CONNECTIONS
    END_SUBAPPLICATION
    EVENT_CONNECTIONS
      StorageSkill.INITO TO TurntableSkill.INIT;
      RobotSetStartParams.SetParams TO RobotSkill.SetStartParam_REQ;
      TurnTableSetStartParams.SetParams TO TurntableSkill.Table_SetStartParam_REQ;
      GripperSkill.INITO TO RobotSkill.INIT;
      TurntableSkill.INITO TO GripperSkill.INIT;
    END_CONNECTIONS
    DATA_CONNECTIONS
      TurnTableSetStartParams.WORD TO TurntableSkill.Table_SetStartParam_IN;
      RobotSetStartParams.WORD TO RobotSkill.Robot_SetStartParam_IN;
    END_CONNECTIONS
  END_APPLICATION
  APPLICATION VDMA_Station1_HierarchicalControl_Distributed
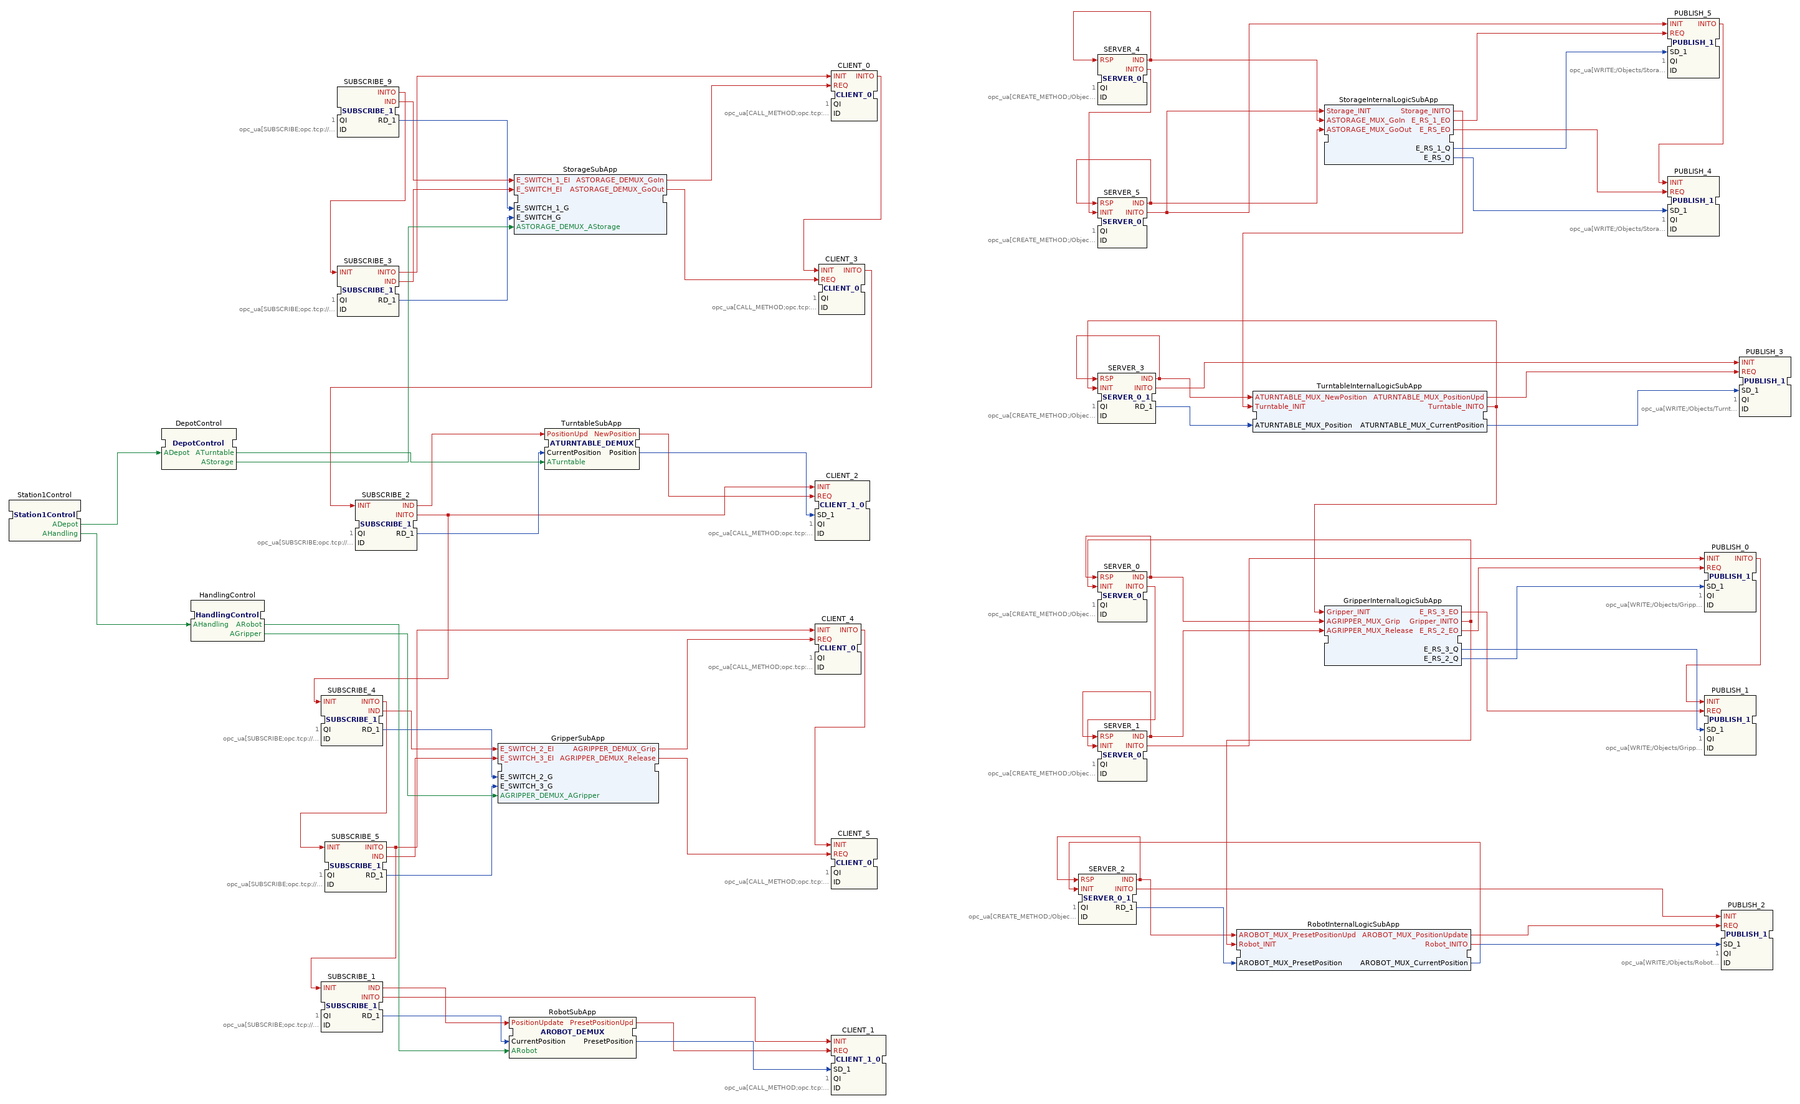
    FBS
      HandlingControl : HandlingControl;
      DepotControl : DepotControl;
      Station1Control : Station1Control;
      SERVER_0 : SERVER_0(QI := 1, ID := opc_ua[CREATE_METHOD;/Objects/Gripper/Grip]);
      SERVER_1 : SERVER_0(QI := 1, ID := opc_ua[CREATE_METHOD;/Objects/Gripper/Release]);
      PUBLISH_2 : PUBLISH_1(QI := 1, ID := opc_ua[WRITE;/Objects/Robot/CurrentPosition]);
      PUBLISH_3 : PUBLISH_1(QI := 1, ID := opc_ua[WRITE;/Objects/Turntable/CurrentPosition]);
      SERVER_4 : SERVER_0(QI := 1, ID := opc_ua[CREATE_METHOD;/Objects/Storage/GoIn,1:s=Storage_GoIn]);
      SERVER_5 : SERVER_0(QI := 1, ID := opc_ua[CREATE_METHOD;/Objects/Storage/GoOut,1:s=Storage_GoOut]);
      CLIENT_5 : CLIENT_0(QI := 1, ID := opc_ua[CALL_METHOD;opc.tcp://localhost:4843#;/Objects/Gripper/Release]);
      CLIENT_0 : CLIENT_0(QI := 1, ID := opc_ua[CALL_METHOD;opc.tcp://localhost:4842#;/Objects/Storage/GoIn]);
      CLIENT_3 : CLIENT_0(QI := 1, ID := opc_ua[CALL_METHOD;opc.tcp://localhost:4842#;/Objects/Storage/GoOut]);
      CLIENT_4 : CLIENT_0(QI := 1, ID := opc_ua[CALL_METHOD;opc.tcp://localhost:4843#;/Objects/Gripper/Grip]);
      SUBSCRIBE_1 : SUBSCRIBE_1(QI := 1, ID := opc_ua[SUBSCRIBE;opc.tcp://localhost:4840#;/Objects/Robot/CurrentPosition]);
      RobotSubApp : AROBOT_DEMUX;
      SUBSCRIBE_2 : SUBSCRIBE_1(QI := 1, ID := opc_ua[SUBSCRIBE;opc.tcp://localhost:4841#;/Objects/Turntable/CurrentPosition]);
      TurntableSubApp : ATURNTABLE_DEMUX;
      PUBLISH_5 : PUBLISH_1(QI := 1, ID := opc_ua[WRITE;/Objects/Storage/IsIn]);
      PUBLISH_4 : PUBLISH_1(QI := 1, ID := opc_ua[WRITE;/Objects/Storage/IsOut]);
      SUBSCRIBE_3 : SUBSCRIBE_1(QI := 1, ID := opc_ua[SUBSCRIBE;opc.tcp://localhost:4842#;/Objects/Storage/IsOut]);
      SUBSCRIBE_9 : SUBSCRIBE_1(QI := 1, ID := opc_ua[SUBSCRIBE;opc.tcp://localhost:4842#;/Objects/Storage/IsIn]);
      PUBLISH_1 : PUBLISH_1(QI := 1, ID := opc_ua[WRITE;/Objects/Gripper/Released]);
      PUBLISH_0 : PUBLISH_1(QI := 1, ID := opc_ua[WRITE;/Objects/Gripper/Gripped]);
      SUBSCRIBE_4 : SUBSCRIBE_1(QI := 1, ID := opc_ua[SUBSCRIBE;opc.tcp://localhost:4843#;/Objects/Gripper/Gripped]);
      SUBSCRIBE_5 : SUBSCRIBE_1(QI := 1, ID := opc_ua[SUBSCRIBE;opc.tcp://localhost:4843#;/Objects/Gripper/Released]);
      SERVER_3 : SERVER_0_1(QI := 1, ID := opc_ua[CREATE_METHOD;/Objects/Turntable/NewPosition]);
      CLIENT_2 : CLIENT_1_0(QI := 1, ID := opc_ua[CALL_METHOD;opc.tcp://localhost:4841#;/Objects/Turntable/NewPosition]);
      CLIENT_1 : CLIENT_1_0(QI := 1, ID := opc_ua[CALL_METHOD;opc.tcp://localhost:4840#;/Objects/Robot/PresetPositionUpd]);
      SERVER_2 : SERVER_0_1(QI := 1, ID := opc_ua[CREATE_METHOD;/Objects/Robot/PresetPositionUpd]);
    END_FBS
    SUBAPPLICATION StorageSubApp
      EVENT_INPUT
        E_SWITCH_1_EI;
        E_SWITCH_EI;
      END_EVENT
      EVENT_OUTPUT
        ASTORAGE_DEMUX_GoIn;
        ASTORAGE_DEMUX_GoOut;
      END_EVENT
      VAR_INPUT
        E_SWITCH_1_G : BOOL;
        E_SWITCH_G : BOOL;
      END_VAR
      SOCKETS
        ASTORAGE_DEMUX_AStorage : AStorage;
      END_SOCKETS
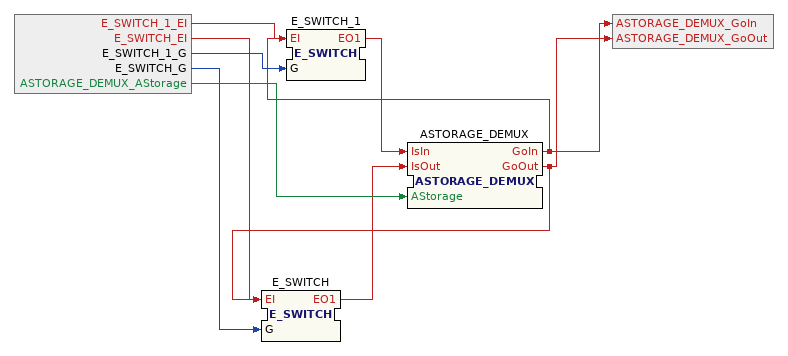
      FBS
        E_SWITCH_1 : E_SWITCH;
        E_SWITCH : E_SWITCH;
        ASTORAGE_DEMUX : ASTORAGE_DEMUX;
      END_FBS
      EVENT_CONNECTIONS
        ASTORAGE_DEMUX.GoIn TO E_SWITCH_1.EI;
        E_SWITCH_1.EO1 TO ASTORAGE_DEMUX.IsIn;
        ASTORAGE_DEMUX.GoOut TO E_SWITCH.EI;
        E_SWITCH.EO1 TO ASTORAGE_DEMUX.IsOut;
        E_SWITCH_1_EI TO E_SWITCH_1.EI;
        E_SWITCH_EI TO E_SWITCH.EI;
        ASTORAGE_DEMUX.GoIn TO ASTORAGE_DEMUX_GoIn;
        ASTORAGE_DEMUX.GoOut TO ASTORAGE_DEMUX_GoOut;
      END_CONNECTIONS
      DATA_CONNECTIONS
        E_SWITCH_1_G TO E_SWITCH_1.G;
        E_SWITCH_G TO E_SWITCH.G;
      END_CONNECTIONS
      ADAPTER_CONNECTIONS
        ASTORAGE_DEMUX_AStorage TO ASTORAGE_DEMUX.AStorage;
      END_CONNECTIONS
    END_SUBAPPLICATION
    SUBAPPLICATION GripperSubApp
      EVENT_INPUT
        E_SWITCH_2_EI;
        E_SWITCH_3_EI;
      END_EVENT
      EVENT_OUTPUT
        AGRIPPER_DEMUX_Grip;
        AGRIPPER_DEMUX_Release;
      END_EVENT
      VAR_INPUT
        E_SWITCH_2_G : BOOL;
        E_SWITCH_3_G : BOOL;
      END_VAR
      SOCKETS
        AGRIPPER_DEMUX_AGripper : AGripper;
      END_SOCKETS
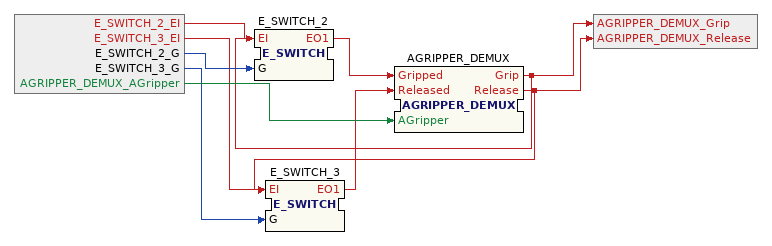
      FBS
        E_SWITCH_2 : E_SWITCH;
        AGRIPPER_DEMUX : AGRIPPER_DEMUX;
        E_SWITCH_3 : E_SWITCH;
      END_FBS
      EVENT_CONNECTIONS
        AGRIPPER_DEMUX.Grip TO E_SWITCH_2.EI;
        E_SWITCH_2.EO1 TO AGRIPPER_DEMUX.Gripped;
        E_SWITCH_3.EO1 TO AGRIPPER_DEMUX.Released;
        AGRIPPER_DEMUX.Release TO E_SWITCH_3.EI;
        E_SWITCH_2_EI TO E_SWITCH_2.EI;
        AGRIPPER_DEMUX.Grip TO AGRIPPER_DEMUX_Grip;
        AGRIPPER_DEMUX.Release TO AGRIPPER_DEMUX_Release;
        E_SWITCH_3_EI TO E_SWITCH_3.EI;
      END_CONNECTIONS
      DATA_CONNECTIONS
        E_SWITCH_2_G TO E_SWITCH_2.G;
        E_SWITCH_3_G TO E_SWITCH_3.G;
      END_CONNECTIONS
      ADAPTER_CONNECTIONS
        AGRIPPER_DEMUX_AGripper TO AGRIPPER_DEMUX.AGripper;
      END_CONNECTIONS
    END_SUBAPPLICATION
    SUBAPPLICATION StorageInternalLogicSubApp
      EVENT_INPUT
        Storage_INIT;
        ASTORAGE_MUX_GoIn;
        ASTORAGE_MUX_GoOut;
      END_EVENT
      EVENT_OUTPUT
        Storage_INITO;
        E_RS_1_EO;
        E_RS_EO;
      END_EVENT
      VAR_OUTPUT
        E_RS_1_Q : BOOL;
        E_RS_Q : BOOL;
      END_VAR
